FUNCTION_BLOCK PUBLIC ACMethodVacuum EXTENDS ACMethodRouteBase
VAR_INPUT
END_VAR
VAR_OUTPUT
END_VAR
VAR PERSISTENT
	_Parameter : ACMethodVacuumP;
	_Result : ACMethodVacuumR;
END_VAR

PROPERTY IsValid : BOOL
GET
IsValid := TRUE;
END_GET
END_PROPERTY

PROPERTY Parameter : ACMethodVacuumP
GET
Parameter := _Parameter;
END_GET
SET // PUBLIC
_Parameter := Parameter;
END_SET
END_PROPERTY

PROPERTY Result : ACMethodVacuumR
GET
Result := _Result;
END_GET
SET // PUBLIC
_Result := Result;
END_SET
END_PROPERTY

END_FUNCTION_BLOCK

(* stored: Version 1.1.0.1, ProductVersion 3.1.4020.12
   POU ACMethodVacuum: Id {6b4933e1-f730-446f-a666-d70106d0291a}, SpecialFunc None
   Property IsValid: Id {aae50082-92ab-454e-98f0-abf59943cb27}
   Get Get: Id {37611b0d-e248-4e41-b154-8cc0041f0cb9}
   Property Parameter: Id {5cdd3dec-8957-41bd-a52c-ebe93b73df41}
   Get Get: Id {32b17611-5c74-4287-a514-ead9199e94dc}
   Set Set: Id {5d98b568-deee-4bc0-9671-f893954c7425}
   Property Result: Id {efaabf01-a49c-4087-b034-85810509a63a}
   Get Get: Id {777b8b85-0ee0-4d2b-9bae-552be9f3b145}
   Set Set: Id {f7a9d232-0a9b-4eb2-844b-86cf067e847d} *)
